{attribute 'enable_dynamic_creation'}
FUNCTION_BLOCK FB_Nozzle EXTENDS FB_PieceBase
VAR_INPUT
END_VAR
VAR_OUTPUT
END_VAR
VAR
	nCleaningDepth	: DINT;
END_VAR

METHOD FB_init : BOOL
VAR_INPUT
	bInitRetains : BOOL; // if TRUE, the retain variables are initialized (warm start / cold start)
	bInCopyCode : BOOL;  // if TRUE, the instance afterwards gets moved into the copy code (online change)
END_VAR
eObjectType := E_ObjectType.OBJECTTYPE_Nozzle;
eObjectGroup := E_ObjectGroup.OBJECTGROUP_Piece;
END_METHOD

METHOD M_GetAllProps : ERRORID
VAR_INPUT
	refCmdData : REFERENCE TO  ST_CmdData;
END_VAR
SUPER^.M_GetAllProps(refCmdData);
nCurrentPropIndex := nCurrentPropIndex + 1;
refCmdData.n32Data[nCurrentPropIndex] := nCleaningDepth;
END_METHOD

{attribute 'object_name' := 'M_SetAllProps'}
METHOD M_SetAllProps : ERRORID
VAR_INPUT
	refCmdData	: REFERENCE TO ST_CmdData;
END_VAR
M_SetAllProps := SUPER^.M_SetAllProps(refCmdData);

IF M_SetAllProps > 0 THEN
	RETURN;
END_IF
nCurrentPropIndex := nCurrentPropIndex + 1;
nSpecPropIndex := nCurrentPropIndex;

nCleaningDepth := refCmdData.n32Data[nCurrentPropIndex];

nNoOfProps := nCurrentPropIndex + 1;
END_METHOD

METHOD M_SetSingleProp : ERRORID
VAR_INPUT
	refCmdData : REFERENCE TO  ST_CmdData;
END_VAR
IF refCmdData.aHeader[1] = nSpecPropIndex THEN
	nCleaningDepth := refCmdData.n32Data[0];	
ELSE
	M_SetSingleProp := SUPER^.M_SetSingleProp(refCmdData);
END_IF
END_METHOD

PROPERTY P_nCleaningDepth : DINT
GET
P_nCleaningDepth := nCleaningDepth;
END_GET
END_PROPERTY

END_FUNCTION_BLOCK

(* stored: Version 1.1.0.1, ProductVersion 3.1.4022.18
   POU FB_Nozzle: Id {88899545-ff27-4717-82e8-59085e3ccbd0}, SpecialFunc None
   Method FB_init: Id {cc1116ac-acf7-427e-a754-2ce7957ea169}
   Method M_GetAllProps: Id {f1b32e47-7fe4-4869-a36a-23f8b894b70f}
   Method M_SetAllProps: Id {018a72ac-11fb-4e29-9218-b3315dafa34d}
   Method M_SetSingleProp: Id {7a494432-71cb-42ee-9222-9660adc0cba2}
   Property P_nCleaningDepth: Id {88b4fe02-0413-4edd-9a6e-a235da167c47}
   Get Get: Id {67e948a0-cba4-478f-bd61-fdc41938a2c7} *)
